{attribute 'GeneratedUsingTerminal: EK1100-0000-0018'}
{attribute addProperty BoxType "EK1100-0000-0018"}
{attribute addProperty Id "Term_154_EK1122Term_154_EK1122_E57516AE40Term_155_EL2008EL2008_E2806B9511Term_156_EL2008EL2008_E2806B9511"}
{attribute addProperty CRC "2445327176"}
{attribute addProperty Size "62"}
{attribute addProperty Name "Term 153 (EK1100)"}
TYPE Term_153_EK1100_91C0BB48 EXTENDS EK1100_1FC0878B :
STRUCT
	{attribute addProperty Name "Term 154 (EK1122)"}
	{attribute addProperty PreviousPort "Term 153 (EK1100) : B"}
	{attribute addProperty SyncUnit "default"}
	Term_154_EK1122 : Term_154_EK1122_E57516AE;
	{attribute addProperty Name "Term 155 (EL2008)"}
	{attribute addProperty PreviousPort "Term 154 (EK1122) : C"}
	{attribute addProperty SyncUnit "default"}
	Term_155_EL2008 : EL2008_E2806B95;
	{attribute addProperty Name "Term 156 (EL2008)"}
	{attribute addProperty PreviousPort "Term 155 (EL2008) : B"}
	{attribute addProperty SyncUnit "default"}
	Term_156_EL2008 : EL2008_E2806B95;
END_STRUCT
END_TYPE

(* stored: Version 1.2.0.0, ProductVersion 3.1.4024.11
   DUT Term_153_EK1100_91C0BB48: Id {62394f70-2e00-4b39-bb85-6781766d909b} *)
